// TIA Portal V19 export
VAR_GLOBAL   // PLC tag table "Sorties"
   "1M2" AT %Q0.0 : Bool;   // Descente vérin élévation pièce
   "1M1" AT %Q0.1 : Bool;   // Montée vérin élévation pièce
   "2M1" AT %Q0.2 : Bool;   // Sortie vérin éjection pièce
   "3M1" AT %Q0.3 : Bool;   // Activation toboggan pneumatique
   LStart AT %Q1.0 : Bool;   // Lampe BP Start
   LReset AT %Q1.1 : Bool;   // Lampe BP Reset
   Q1 AT %Q1.2 : Bool;   // Voyant lumineux Q1
   Q2 AT %Q1.3 : Bool;   // Voyant lumineux Q2
END_VAR
